INTERFACE I_VarByteBufferBase

PROPERTY Buffer : PVOID
GET
END_GET
END_PROPERTY

PROPERTY Capacity : UDINT
GET
END_GET
END_PROPERTY

METHOD Clear : BOOL
END_METHOD

PROPERTY FreeBytes : UDINT
GET
END_GET
END_PROPERTY

METHOD Initialize : BOOL
VAR_INPUT
	nBufferSize 		: UDINT; // Size in byte
END_VAR
END_METHOD

METHOD Reset
END_METHOD

PROPERTY Size : UDINT
GET
END_GET
END_PROPERTY

END_INTERFACE

(* stored: Version 1.1.0.1
   Itf I_VarByteBufferBase: Id {5621949c-0dc6-457e-b23e-0aa68299a226}
   Property Buffer: Id {ce02aefb-10a8-4021-8369-7d6fe79ae8ed}
   Get Get: Id {68add254-d745-4efa-b43a-6be5f717727d}
   Property Capacity: Id {90e1910c-1e1b-4944-974f-e8ad2db93c4a}
   Get Get: Id {d610a920-f74d-4fc0-a47e-80414dbca44b}
   Method Clear: Id {2d19adf6-cb85-4b7b-ad1b-09b498e54220}
   Property FreeBytes: Id {beb246ef-0add-4f7a-8a6c-5ce94ef3d7f8}
   Get Get: Id {03dde9c7-e630-4f22-96e8-b312278bb7d4}
   Method Initialize: Id {37837a7f-e622-4fa7-be59-3210f83b4fe5}
   Method Reset: Id {c42e50a3-a6c0-44d8-8679-cf6cdca02325}
   Property Size: Id {055fb05f-bc3d-43b5-bc16-baeee001edf2}
   Get Get: Id {5dd2b769-789e-41fa-84af-4288920eb036} *)
